FUNCTION_BLOCK L6_plosina_FBD
VAR_INPUT
	TL: BOOL;
	CPL: BOOL;
	CPE0: BOOL;
	CPE1: BOOL;
	CPD0: BOOL;
	CPD1: BOOL;
END_VAR
VAR_OUTPUT
	RPE0: BOOL;
	RPE1: BOOL;
	RPD: BOOL;
END_VAR
VAR
END_VAR

// NETWORK 1

END_FUNCTION_BLOCK

(* stored: Version 1.1.0.1, ProductVersion 3.1.4024.13
   POU L6_plosina_FBD: Id {d24d1f36-7618-4396-88b9-00ed89815f18}, SpecialFunc None *)
